{attribute 'linkalways'} 
{attribute 'no_explicit_call' := 'This FB is a CLASS and must be accessed using methods or properties'}
{attribute 'enable_dynamic_creation'}
FUNCTION_BLOCK JsonPathElement_Root EXTENDS JsonPathElement 
VAR
END_VAR

PROPERTY PUBLIC PropertyName : T_MAXSTRING
GET
PropertyName := 'root';
END_GET
END_PROPERTY

METHOD PUBLIC ResolveToSJsonValue : SJsonValue
VAR_INPUT
	jsonParser : REFERENCE TO FB_JsonDomParser;
	jsonDocument : SJsonValue;
END_VAR
ResolveToSJsonValue := jsonDocument;
END_METHOD

END_FUNCTION_BLOCK

(* stored: Version 1.1.0.1, ProductVersion 3.1.4024.12
   POU JsonPathElement_Root: Id {4040b4a2-0a3f-0e0c-26c7-535ab52052ee}, SpecialFunc None
   Property PropertyName: Id {923a460c-e872-09c8-1027-12658d5ac8d2}
   Get Get: Id {e3e4527e-8faa-0f01-1f86-589d368b3fd6}
   Method ResolveToSJsonValue: Id {73905360-aeb4-05e6-0325-b1873e748940} *)
